FUNCTION_BLOCK AB2_TO_AB (* Composite FB for convert bidirectional AB2 to unidirectional AB *)
  (* Standard: 61499-2; Function: AB2_BIDIR forwards its incoming (EO1) side out as a plain unidirectional signal via AB_OUT. AB_IN publishes its value onto the outgoing (EI1) side of AB2_BIDIR.; Description: Copyright (c) 2026 HR Agrartechnik GmbH This program and the accompanying materials are made available under the terms of the Eclipse Public License 2.0 which is available at https://www.eclipse.org/legal/epl-2.0/ SPDX-License-Identifier: EPL-2.0 *)
  (* Version 1.0, 2026-08-31, Franz Höpfinger, HR Agrartechnik GmbH, Initial Version *)
  PACKAGE adapter::conversion::bidirectional;
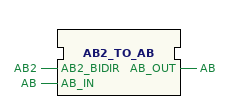
  SOCKETS
    AB2_BIDIR : adapter::types::bidirectional::AB2; (* Adapter Input: bidirectional tap, incoming side forwarded to AB_OUT, outgoing side driven by AB_IN *)
    AB_IN : adapter::types::unidirectional::AB; (* Adapter Input: unidirectional source *)
  END_SOCKETS
  PLUGS
    AB_OUT : adapter::types::unidirectional::AB; (* Adapter Output: mirrors AB2_BIDIR's incoming (indication) side *)
  END_PLUGS
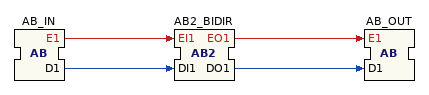
  EVENT_CONNECTIONS
    AB2_BIDIR.EO1 TO AB_OUT.E1;
    AB_IN.E1 TO AB2_BIDIR.EI1;
  END_CONNECTIONS
  DATA_CONNECTIONS
    AB2_BIDIR.DO1 TO AB_OUT.D1;
    AB_IN.D1 TO AB2_BIDIR.DI1;
  END_CONNECTIONS
END_FUNCTION_BLOCK
